(* PLC project Untitled1, Beckhoff Automation GmbH TwinCAT PLC Control 3.5.13.21 *)
(* stored: creationDateTime 2022-05-01T12:16:10.5796063, modificationDateTime 2022-05-01T12:16:10.5796063 *)

FUNCTION_BLOCK FB_McVelocity

VAR_INPUT
	bStart					: BOOL;
	bStop					: BOOL;
	fAxisAccel				: REAL;
	fAxisDecel				: REAL;
	eAxisDirection			: MC_Direction;
	fAxisSpeed				: REAL;
	bReset					: BOOL;
END_VAR

VAR_OUTPUT
	bError					: BOOL;
END_VAR

VAR
	stAxis					: AXIS_REF;
	fbAxisEnable			: MC_Power;
	fbAxisVelocity			: MC_MoveVelocity;
	fbAxisStop				: MC_Stop;
	fbAxisReset				: MC_Reset;
	bTogglePulse			: BOOL;
	fbStart					: R_TRIG;
	fbStop					: R_TRIG;
	eMcVelocityState 		: (WAIT, ENABLE_AXIS, RUN, STOP, DISABLE_AXIS, ERROR);
END_VAR

            fbStart(CLK := bStart);
fbStop(CLK := bStop);
bTogglePulse := NOT bTogglePulse;
stAxis.ReadStatus();

CASE eMcVelocityState OF
	
	WAIT:
	
		IF fbStart.Q AND NOT fbStop.Q THEN
			fbAxisStop(Axis := stAxis, Execute := FALSE);
			eMcVelocityState := ENABLE_AXIS;
		END_IF
		
		
	ENABLE_AXIS:
		
		fbAxisEnable(Axis := stAxis,
			  Enable := TRUE,
			  Enable_Positive := TRUE,
			  Enable_Negative := TRUE,
			  Override := 100);
			  
		IF stAxis.Status.Operational AND NOT fbStop.Q THEN
			eMcVelocityState := RUN;
		ELSIF stAxis.Status.Operational AND fbStop.Q THEN
			eMcVelocityState := DISABLE_AXIS;
		ELSIF stAxis.Status.Error THEN
			eMcVelocityState := ERROR;
		END_IF
	
		
	RUN:
	
		fbAxisVelocity(
			Axis         := stAxis,
			Execute      := bTogglePulse,
			Acceleration := fAxisAccel,
			Deceleration := fAxisDecel,
			Direction    := eAxisDirection,
			BufferMode   := MC_BufferMode.MC_Aborting,
			Velocity     := fAxisSpeed
			);
		
		IF stAxis.Status.Operational AND fbStop.Q THEN
			eMcVelocityState := STOP;
		ELSIF stAxis.Status.Error THEN
			eMcVelocityState := ERROR;
		END_IF
		
		
	STOP:
		
		fbAxisStop(			
			Axis         := stAxis,
			Execute      := TRUE,
			Deceleration := fAxisDecel,
			);
	
		IF stAxis.Status.NotMoving THEN
			eMcVelocityState := DISABLE_AXIS;
		END_IF
			
	
	DISABLE_AXIS:
	
		fbAxisEnable(
			Axis := stAxis,
			Enable := FALSE,
			Enable_Positive := FALSE,
			Enable_Negative := FALSE,
			Override := 0);
			 
		IF stAxis.Status.Disabled AND NOT stAxis.Status.Error THEN
			eMcVelocityState := WAIT;
		ELSIF stAxis.Status.Disabled AND stAxis.Status.Error THEN
			eMcVelocityState := ERROR;
		END_IF
	
		
	ERROR:
	
		bError := TRUE;
		
		IF bReset THEN
			fbAxisReset(
				Axis := stAxis, 
				Execute := TRUE);
			IF NOT stAxis.Status.Error THEN
				bError := FALSE;
				fbAxisReset(
					Axis := stAxis, 
					Execute := FALSE);
				eMcVelocityState := WAIT;
			END_IF
		END_IF
		
END_CASE


			  
		
          
END_FUNCTION_BLOCK
